{attribute 'pack_mode' := '1'}
TYPE ST_CanData_11bit :
STRUCT
	nCobid: WORD; //bits 0-3 is CAN data length, bit 4 is CAN RTR flag, bit 5-15 is CAN Cobid.
	aData: ARRAY[0..7] OF BYTE;
END_STRUCT
END_TYPE

(* stored: Version 1.1.0.1, ProductVersion 3.1.4024.11
   DUT ST_CanData_11bit: Id {9ede8b97-692a-4df0-8347-39337e51bfb4} *)
